Staubli VAL3: libGeneric_0_1.pjx

--- libGeneric_0_1.pjx ---
Parameters version=s7.7.2 stackSize=5000 millimeterUnit=true
Program file=empty1dNum.pgx
Program file=empty2dNum.pgx
Program file=merge1dNum.pgx
Program file=shiftArray.pgx
Program file=trimAsciiBuffer.pgx
Data file=libGeneric_0_1.dtx

--- empty1dNum.pgx ---
public program empty1dNum(num& x_nNum[])
  local num l_nIndex
begin

  //empty a 1d array of num

  for l_nIndex=0 to size(x_nNum)-1
      x_nNum[l_nIndex]=0
  endFor

end

--- merge1dNum.pgx ---
public program merge1dNum(num& x_nNum1[], num& x_nNum2[], num& x_nMerged[])
  local num l_nIndex
  local num i
begin

  resize(x_nMerged,1,size(x_nNum1)+size(x_nNum2))
  call empty1dNum(x_nMerged)

  for l_nIndex=0 to size(x_nNum1)-1
    x_nMerged[i]=x_nNum1[l_nIndex]
    i=i+1
  endFor

  for l_nIndex=0 to size(x_nNum2)-1
    x_nMerged[i]=x_nNum2[l_nIndex]
    i=i+1
  endFor

end
